{attribute 'qualified_only'}
{attribute 'strict'}
TYPE E_SocketSendState :
(
	READY,
	SENDING,
	DONE,
	ERROR
);
END_TYPE

(* stored: Version 1.1.0.1, ProductVersion 3.1.4024.13
   DUT E_SocketSendState: Id {a3093089-5b91-4893-a49f-486517aeda48} *)
